PROGRAM PGRTestFB
VAR
	Fb_Calculate : FB_CalCulateAccumulation;
	lrAccumulation : LREAL;
	CurrentTime : TIMESTRUCT;
	previoustime : TIMESTRUCT;
	bAcknowledgeNewPeriodAlarm : BOOL ;
	bMRAckAlarm	: BOOL;
	Value1Minute : LREAL;
	value1Hour	: LREAL;
	value1Day : LREAL;
	bEventHour : BOOL;
	bEventDay : BOOL;
	bFirstCycle : BOOL := TRUE;
	bReset	: BOOL;
	eTimeAccumulate : E_CompareTime;
	

END_VAR
VAR
	fbFIFO_lr : FB_FIFO_Lreal;
	bFull : BOOL;
	bempty : BOOL;
	valueOut : LREAL;
	ValueInt : LREAL;
	ackValue : BOOL;
	Addvalue : BOOL;
	ResetFIFO : BOOL;
	head : UINT;
	Tail : UINT;
	Nt_systemTime : TIMESTRUCT;
	fb_localsystemtime : TIMESTRUCT;
	
END_VAR

///
	lrAccumulation := lrAccumulation + 0.01;
	
	Fb_Calculate.TimeAccumulate := eTimeAccumulate;
	
	IF bFirstCycle THEN
		 IF Fb_Calculate.MR_Init() THEN bFirstCycle := FALSE; END_IF;
	END_IF
	
	Fb_Calculate(lrAccumulator := lrAccumulation,
					accumulatedValueOut => Value1Minute,
					previousTimestampOut => previoustime,
					bNewPeriodAlarm => bAcknowledgeNewPeriodAlarm);
					
	IF bMRAckAlarm THEN 
		IF Fb_Calculate.MR_Acknowledge() THEN
			bMRAckAlarm := FALSE ; 
		END_IF
	END_IF
	IF bReset THEN
		IF Fb_Calculate.MR_Reset() THEN
			bReset := FALSE;
		END_IF
	END_IF
/////////

bempty :=	fbFIFO_lr.IsEmpty;
bFull := fbFIFO_lr.IsFull;

IF ackValue THEN
	IF fbFIFO_lr.MR_AckGetValue() THEN
		ackValue := FALSE;
	END_IF
END_IF		

IF Addvalue THEN
	IF fbFIFO_lr.MR_AddValue( Value := ValueInt)THEN
		Addvalue := FALSE;
	END_IF
END_IF

IF ResetFIFO THEN
	IF fbFIFO_lr.MR_Reset() THEN
		ResetFIFO := FALSE;
	END_IF
END_IF
valueOut := fbFIFO_lr.OldestData;
head := fbFIFO_lr.HeadIndex;
Tail := fbFIFO_lr.TailIndex;
///
Nt_systemTime := pmDev.NT_GetTime.TIMESTR;
fb_localsystemtime := GVL.fbMachineTime.systemTime;

END_PROGRAM

(* stored: Version 1.1.0.1, ProductVersion 3.1.4024.12
   POU PGRTestFB: Id {206e4f68-a63b-4760-bf2b-dfc0027728aa}, SpecialFunc None *)
